// TIA Portal project "Üretim Hattı Factory.io'da Pano Kullanımı_V15.1" (V15.1)
// Vorlageprojekt für das Buch mit Zielsystem S7-1200

(* hardware
DEVICE "S7-1200-Station_1"  S7-1200 Station
   slot 0: "Baugruppenträger_0"  Rack  V1.0
   slot 1: "PLC_1"  CPU 1211C DC/DC/DC  6ES7 211-1AE40-0XB0  V4.1
DEVICE "PC-System_1"  SIMATIC PC station
   slot 0: "SIMATIC PC station"  Rail  SIMATIC PC-Station  V1.0
      slot 125: "Stationmanager"  Station_Manager  V6.0.4
   slot 1: "HMI_RT_1"  WinCC RT Advanced  6AV2 104-0xxxx-xxxx  15.1.0.0
      slot 33792: "Host interface"  Host interface
   slot 2: "IE general_1"  IE General  IE_CP  V8.2.0
*)

// ===== PLC "PLC_1"  CPU 1211C DC/DC/DC =====

VAR_GLOBAL   // PLC tag table "plc_tags"
   "stop" AT %I0.0 : Bool;
   "start" AT %I0.1 : Bool;
   "sistem_devrede" AT %M5.0 : Bool;
   "yardimci_mem" AT %M5.1 : Bool;
   "sistem_lambasi" AT %Q0.0 : Bool;
   "konvenyör" AT %Q0.1 : Bool;
END_VAR

VAR_GLOBAL   // PLC tag table "hmi_tags"
   "HMI_start" AT %M6.0 : Bool;
   "HMI_stop" AT %M6.1 : Bool;
   "HMI_lamba" AT %M6.2 : Bool;
   "hmi_kutuyu_kaydir" AT %QW1 : Int;
END_VAR

FUNCTION "MHJ-PLC-Lab-Function-S71200" : Void   // FC9000, SCL
{ S7_Optimized_Access := 'TRUE' }
VERSION : 0.1
   VAR_TEMP
      rdTimeReturn : Int;
      outputTime : DTL;
      SyncVal : Byte;
      forVal : Int;
      forVal_2 : Int;
      Value : Byte;
   END_VAR
   VAR CONSTANT
      CompVal : Byte := 16#34;
      Value_01 : Byte := 16#11;
      Value_01_DW : DWord := 16#A165_D992;
      Value_02_DW : DWord := 16#58BE_4401;
   END_VAR
BEGIN

   #Value:=PEEK(area := 16#82,
        dbNumber := 0,
        byteOffset := 511);
   #Value := #Value + 1;

   POKE(area := 16#82,
        dbNumber := 0,
        byteOffset := 511,
        value := #Value);

   POKE(area:=16#81,
        dbNumber:=0,
        byteOffset:=1016,
        value:=#Value_01_DW);
   POKE(area := 16#81,
        dbNumber := 0,
        byteOffset := 1020,
        value := #Value_02_DW);

   POKE(area := 16#81,
        dbNumber := 0,
        byteOffset := 511,
        value := B#16#00);

   FOR #forVal := 0 TO 120 DO
       FOR #forVal_2:=0 TO 10 DO
           #rdTimeReturn:=RD_SYS_T(#outputTime);
           #rdTimeReturn := WR_SYS_T(#outputTime);
           #rdTimeReturn := RD_SYS_T(#outputTime);
           #rdTimeReturn := WR_SYS_T(#outputTime);
       END_FOR;
       #SyncVal:= PEEK(area := 16#81,
                      dbNumber := 0,
                      byteOffset := 511);
       IF #SyncVal = #CompVal THEN
          GOTO M_1;
       END_IF;
   END_FOR;
   RETURN;

   M_1:
   POKE(area := 16#81,
        dbNumber := 0,
        byteOffset := 511,
        value := B#16#0);
END_FUNCTION

ORGANIZATION_BLOCK "Main"   // OB1, LAD, ProgramCycle
TITLE = "Main Program Sweep (Cycle)"
{ S7_Optimized_Access := 'TRUE' }
VERSION : 0.1
   VAR_INPUT
      Initial_Call : Bool;   // Initial call of this OB
      Remanence : Bool;   // =True, if remanent data are available
   END_VAR
   VAR_TEMP
      setreset : Bool;
   END_VAR
BEGIN

REGION Network 1: Konnektierungsbaustein für PLC-Lab
   // Im Netzwerk 1 wird der Konnektierungsbaustein für PLC-Lab aufgerufen.
   // Dieser Aufruf darf nicht entfernt werden!
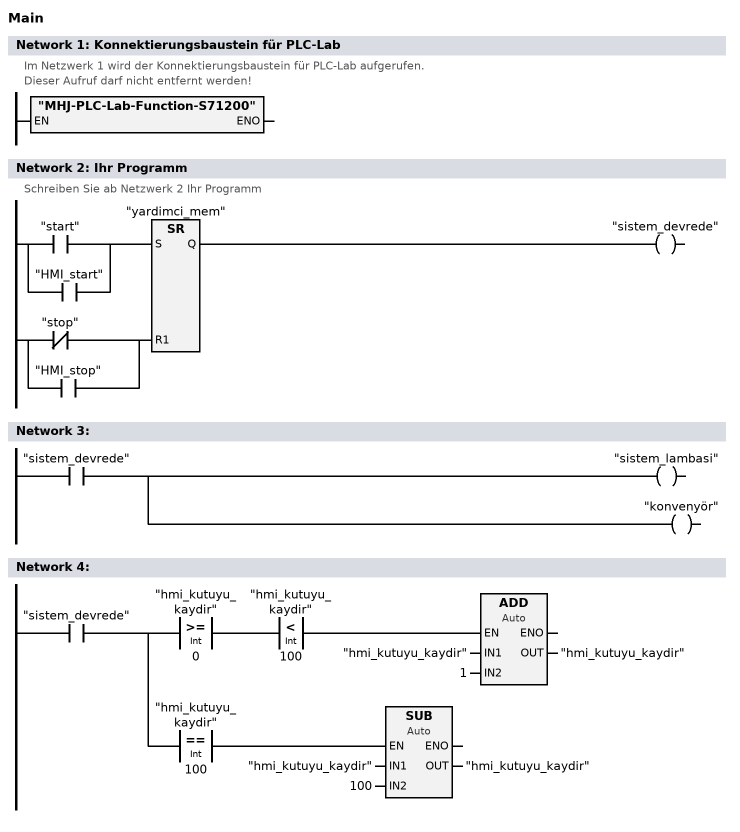
   RUNG wire#powerrail
      "MHJ-PLC-Lab-Function-S71200"()
   END_RUNG
   // the same network as SCL:
   "MHJ-PLC-Lab-Function-S71200"();
END_REGION

REGION Network 2: Ihr Programm
   // Schreiben Sie ab Netzwerk 2 Ihr Programm
   RUNG wire#powerrail
      Contact( "start" )
      wire#w1
      S_SR(operand := "yardimci_mem", r1 := wire#w2)
      Coil( "sistem_devrede" )
   END_RUNG
   RUNG wire#powerrail
      Contact( "HMI_start" )
   END_RUNG wire#w1
   RUNG wire#powerrail
      I_Contact( "stop" )
   END_RUNG wire#w2
   RUNG wire#powerrail
      Contact( "HMI_stop" )
   END_RUNG wire#w2
   // the same network as SCL:
   IF "start" OR "HMI_start" THEN
       "yardimci_mem" := TRUE;   // SR flip-flop
   END_IF;
   IF NOT "stop" OR "HMI_stop" THEN "yardimci_mem" := FALSE; END_IF;
   "sistem_devrede" := "yardimci_mem";
END_REGION

REGION Network 3
   RUNG wire#powerrail
      Contact( "sistem_devrede" )
      wire#w1
      Coil( "sistem_lambasi" )
   END_RUNG
   RUNG wire#w1
      Coil( "konvenyör" )
   END_RUNG
   // the same network as SCL:
   "sistem_lambasi" := "sistem_devrede";
   "konvenyör" := "sistem_devrede";
END_REGION

REGION Network 4
   RUNG wire#powerrail
      Contact( "sistem_devrede" )
      wire#w1
      { S7_Templates := "SrcType := Int" } GE_Contact(in1 := "hmi_kutuyu_kaydir", in2 := 0)
      { S7_Templates := "SrcType := Int" } LT_Contact(in1 := "hmi_kutuyu_kaydir", in2 := 100)
      Add(in1 := "hmi_kutuyu_kaydir", in2 := 1, out => "hmi_kutuyu_kaydir")
   END_RUNG
   RUNG wire#w1
      { S7_Templates := "SrcType := Int" } EQ_Contact(in1 := "hmi_kutuyu_kaydir", in2 := 100)
      Sub(in1 := "hmi_kutuyu_kaydir", in2 := 100, out => "hmi_kutuyu_kaydir")
   END_RUNG
   // the same network as SCL:
   IF "sistem_devrede" AND ("hmi_kutuyu_kaydir" >= 0) AND ("hmi_kutuyu_kaydir" < 100) THEN
       "hmi_kutuyu_kaydir" := "hmi_kutuyu_kaydir" + 1;
   END_IF;
   IF "sistem_devrede" AND ("hmi_kutuyu_kaydir" = 100) THEN
       "hmi_kutuyu_kaydir" := "hmi_kutuyu_kaydir" - 100;
   END_IF;
END_REGION
END_ORGANIZATION_BLOCK

(* ===== HMI "HMI_RT_1" =====
system functions are stored by id; their names below are inferred from use
connection "HMI_Connection_1": ETHERNET, S7_1200_OMS

HMI tags "Default tag table"
   "HMI_start" : Bool = PLC HMI_start AT %M6.0, 100 ms
   "HMI_stop" : Bool = PLC HMI_stop AT %M6.1, 100 ms
   "HMI_lamba" : Bool = PLC HMI_lamba AT %M6.2, 100 ms
   "sistem_lambasi" : Bool = PLC sistem_lambasi AT %Q0.0, 1 s
   "hmi_kutuyu_kaydir" : Int = PLC hmi_kutuyu_kaydir AT %QW1, 1 s

screen "Ana Ekran" 600x800
   Button "Button_1" at 45,163 size 96x32; TextOff 'START'
      on Press: SetBit("HMI_start")
      on Release: ResetBit("HMI_start")
   Button "Button_2" at 45,219 size 96x32; TextOff 'STOP'
      on Press: SetBit("HMI_stop")
      on Release: ResetBit("HMI_stop")
   GraphicView "Graphic view_2" at 163,137 size 300x300; Picture "Graphic_2"
   GraphicView "Graphic view_1" at 279,296 size 73x108; Picture "Graphic_1"
   Circle "Circle_1" at 283,303 size 34x34
      Appearance <- "sistem_lambasi"
   TextField "Text field_1" at 147,47 size 326x39; Text 'KONVENYÖR SİSTEMİ'
   GraphicView "Graphic view_3" at 178,163 size 90x95; Picture "Graphic_3"
      HorizontalMovement <- "hmi_kutuyu_kaydir"
*)